// SIMATIC S7-200 project (STEP 7-Micro/WIN), CPU 224 REL 01.11

SYMBOL_TABLE USER1
B_For            I0.0
B_Rev            I0.1
P_Stop           I0.2
Ena              Q0.0
Forr             Q0.1
Rev              Q0.2
END_SYMBOL_TABLE

ORGANIZATION_BLOCK MAIN:OB1
TITLE=PROGRAM COMMENTS
BEGIN
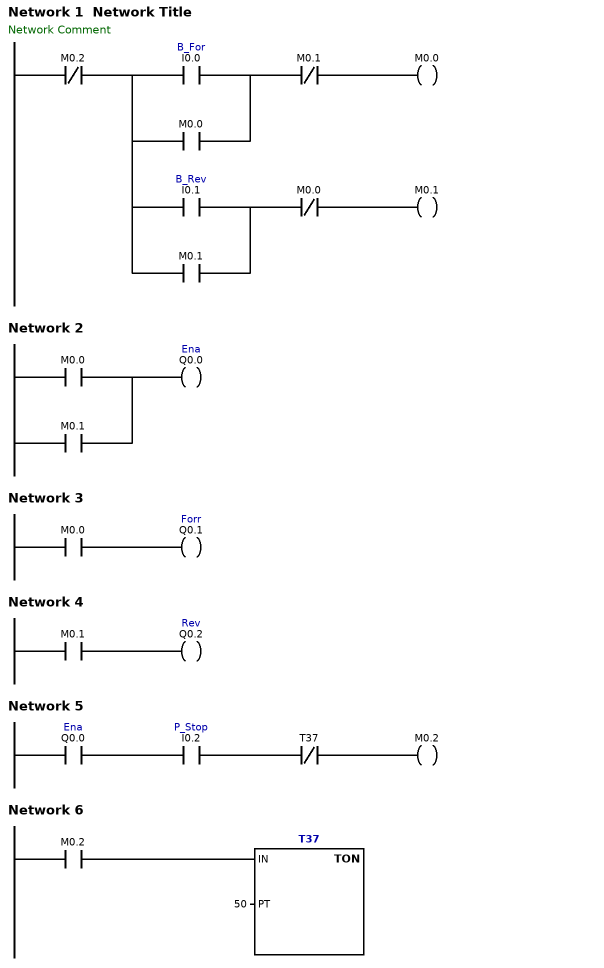
Network 1 // Network Title
// Network Comment
LDN    M0.2
LPS
LD     B_For:I0.0
O      M0.0
ALD
AN     M0.1
=      M0.0
LPP
LD     B_Rev:I0.1
O      M0.1
ALD
AN     M0.0
=      M0.1
Network 2
LD     M0.0
O      M0.1
=      Ena:Q0.0
Network 3
LD     M0.0
=      Forr:Q0.1
Network 4
LD     M0.1
=      Rev:Q0.2
Network 5
LD     Ena:Q0.0
A      P_Stop:I0.2
AN     T37
=      M0.2
Network 6
LD     M0.2
TON    T37, 50
END_ORGANIZATION_BLOCK
